// Gets the size of an object in static memory via its interface.
// Interface must extend FsI_Unknown.
// NOTE: This is performance intensive. Cyclic use is not recommened.
FUNCTION FsF_GetSize : FsT_Size
VAR_INPUT
	ipInterface : FsI_Unknown;
END_VAR
VAR
	pAddress : FsT_Ptr;
END_VAR

pAddress := FsF_GetAddress(ipInterface);
IF pAddress = 0 THEN RETURN; END_IF
CASE Tc2_System.F_CheckMemoryArea(pAddress, 1) OF
	FsT_MemArea.Static:
		FOR FsF_GetSize := SIZEOF(ipInterface) TO FsParam_Core.INFO_SCAN_SIZE DO
			IF FsF_GetTypeNameByAddress(pAddress, FsF_GetSize) <> '' THEN RETURN; END_IF
			END_FOR
		FsF_GetSize := 0;
	END_CASE

END_FUNCTION

(* stored: Version 1.1.0.1, ProductVersion 3.1.4024.4
   POU FsF_GetSize: Id {1c100f78-8ff8-4e04-bdda-082f777a031f}, SpecialFunc None *)
